// TIA Portal V16 export
// export: Created 2023-03-29T11:03:19.2505961Z, ExportSetting WithDefaults, DisplayName Totally Integrated Automation Portal, DisplayVersion V16 Update 6, DisplayName TIA Portal Version Control Interface, DisplayVersion V16 Update 2, DisplayName TIA Portal Openness, DisplayVersion V16 Update 6, DisplayName STEP 7 Professional, DisplayVersion V16 Update 6, DisplayName STEP 7 Safety, DisplayVersion V16, DisplayName WinCC Advanced, DisplayVersion V16 Update 6
DATA_BLOCK "FB220_TimeSyn_PLC_To_HMI_DB_1"   // DB78
VERSION : 0.1
// stored: AutoNumber true, DBAccessibleFromOPCUA true, InstanceOfName FB220_TimeSyn_PLC_To_HMI, InstanceOfType FB
"FB220_TimeSyn_PLC_To_HMI"
   // VAR_OUTPUT
   //    PLC_RD_LOC_T : DTL;
   //    PLC_RD_SYS_T : DTL;
   // END_VAR
   // VAR_IN_OUT
   //    AreaPointer_JobMailbox : Array[0..3] of Word;
   //    SetTime : Bool;
   //    SetDate : Bool;
   // END_VAR
   // VAR
   //    Func_RD_LOC_T : DTL;
   //    Ret_Val_RD_LOC_T : Int;
   //    BCD_Hour : Word;
   //    BCD_Minute : Word;
   //    BCD_Second : Word;
   //    BCD_Weekdday : Word;
   //    BCD_Day : Word;
   //    BCD_Month : Word;
   //    BCD32_Year : DWord;
   //    BCD16_Year : Word;
   //    STEP1 : Bool;
   //    STEP2 : Bool;
   //    STEP3 : Bool;
   //    STEP10 : Bool;
   //    STEP11 : Bool;
   //    STEP12 : Bool;
   //    Func_RD_SYS_T : DTL;
   //    Ret_Val_RD_SYS_T : Int;
   // END_VAR
BEGIN
END_DATA_BLOCK
